Universal Robots PolyScope program: Lab_exe_3_3_70.urp

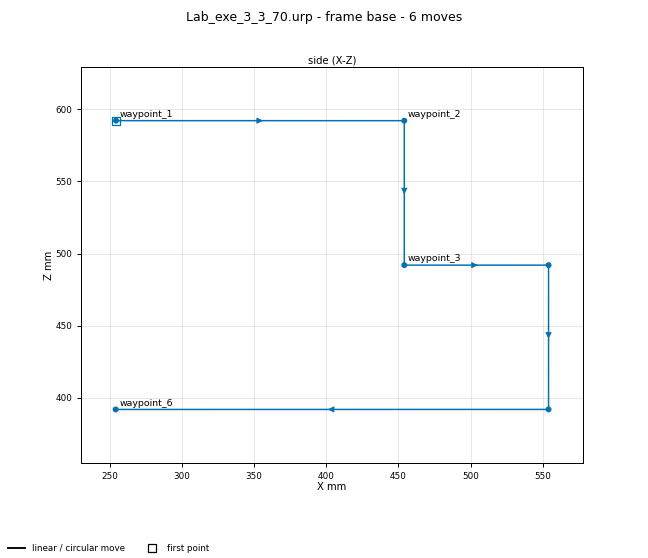
[picture p0: tool path of Lab_exe_3_3_70.urp in frame base, 6 of 6 moves have a stored position in this frame; points joined in program order, loops and branches not executed]
Program Lab_exe_3_3_70 (createdIn=3.2.19293 lastSavedIn=3.2.19293 directory=/programs installation=default robotSerialNumber=2015351391)
Calibrated DH parameters: a=[0.000352, -0.161198, -0.373486, 0.00005, 0.000049, 0]; d=[0.089268, 352.477598, -320.08558, -32.281492, 0.094939, 0.082518]; alpha=[1.570728, 0.001116, -0.003686, 1.571189, -1.570572, 0]; deltaTheta=[-0.000012, 1.181849, -1.491165, 0.309495, -0.000007, 0.000025]
Robot Program (runOnlyOnce=false motionType=MoveJ speed=1.047198 acceleration=1.396263 recalculateMotions=false)
  MoveP speed 250 mm/s, acceleration 1200 mm/s^2 (blendRadius=0.05 recalculateMotions=false) feature=Base
    Waypoint waypoint_1: TCP in base x=254.284 y=198.847 z=592.102 mm, rx=-1.5849 ry=-0.1115 rz=-0.2805 rad; joints [49.675, -69.918, -108.615, -2.42, 124.118, -15.032] deg
    Waypoint waypoint_2: motionParameters(blendRadius=0.05); TCP in base x=454.03 y=198.853 z=592.08 mm, rx=-1.5849 ry=-0.1115 rz=-0.2805 rad; joints [28.741, -97.012, -84.833, 0.384, 145.092, -15.631] deg
    Waypoint waypoint_3: motionParameters(blendRadius=0.05); TCP in base x=454.031 y=198.87 z=491.976 mm, rx=-1.585 ry=-0.1114 rz=-0.2804 rad; joints [28.727, -99.175, -97.196, 14.937, 145.158, -15.59] deg
    Waypoint waypoint_4: motionParameters(blendRadius=0.048); TCP in base x=554.01 y=198.868 z=491.984 mm, rx=-1.5849 ry=-0.1114 rz=-0.2804 rad; joints [23.644, -112.17, -80.279, 10.779, 150.238, -15.845] deg
    Waypoint waypoint_5: TCP in base x=554 y=198.834 z=392.008 mm, rx=-1.5849 ry=-0.1113 rz=-0.2805 rad; joints [23.633, -116.636, -89.204, 24.227, 150.292, -15.781] deg
    Waypoint waypoint_6: TCP in base x=254.017 y=198.864 z=391.982 mm, rx=-1.5852 ry=-0.1112 rz=-0.2804 rad; joints [49.662, -78.21, -133.664, 30.962, 124.243, -14.954] deg
